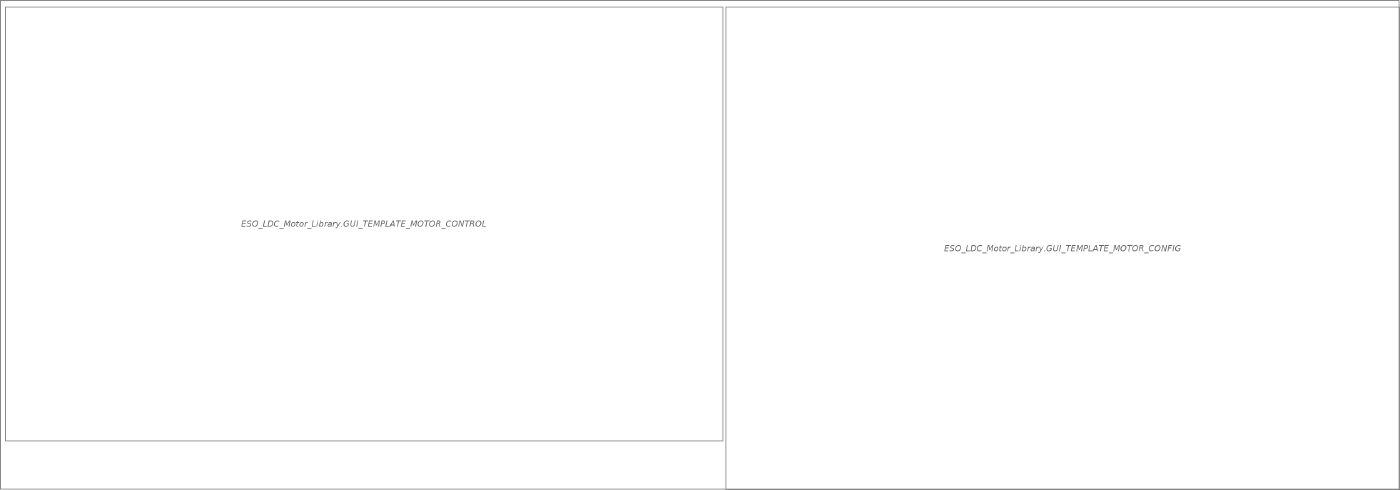
VISUALIZATION GUI_NOTT_DL_1  // 1681x589
    Frame (6,8 862x522)
        shows ESO_LDC_Motor_Library.GUI_TEMPLATE_MOTOR_CONTROL(m_Instance := MAIN.nott_ics.Delay_Lines.NDL1)
    Frame (871,8 810x581)
        shows ESO_LDC_Motor_Library.GUI_TEMPLATE_MOTOR_CONFIG(m_Instance := MAIN.nott_ics.Delay_Lines.NDL1)
END_VISUALIZATION

(* stored: Version 1.1.0.1, ProductVersion 3.1.4024.12
   Visu GUI_NOTT_DL_1: Id {f8bfecd5-0701-4d35-a6f8-9147ddea7056} *)
